TYPE T_CodePO : STRING[20];
END_TYPE

(* stored: Version 1.1.0.1
   DUT T_CodePO: Id {64eb1131-8253-43da-9201-d6a3dd972be3} *)
